FUNCTION_BLOCK FB_TXTDataExchanger IMPLEMENTS I_TXTDataExchanger
VAR CONSTANT
	iBUFFER_SIZE 						: UINT := 255;
END_VAR
VAR
	sName : STRING;
	
	(* First cycle bits used for selecting file logging mode *)
	bAddTimeStamp						: BOOL;
	bAddHeader							: BOOL;
	bCreateFileAtStart					: BOOL;    
                        		
	(* Internal status *)       		
	bActive 							: BOOL;										(*  *)
	bBusy								: BOOL;										(*  *)
	bError								: BOOL;										(*  *)
	iErrorID							: UDINT;									(*  *)
	                                                                            	
	eTXTDataExchangerState 				: E_TXTDataExchangerState;					(*  *)
	eTXTDataExchangerInitState 			: E_TXTDataExchangerInitState;				(*  *)
	eTXTDataExchangerAddLogsState		: E_TXTDataExchangerAddLogsState; 			(*  *)
	eTXTDataExchangerSetNewPathState 	: E_TXTDataExchangerSetNewPathState;
	eTXTDataExchangerSearchForFileState : E_TXTDataExchangerSearchForFileState;
	
	(* Internal parameters *)
	sFileName 							: STRING;									(*  *)
	sFileDir							: STRING;									(*  *)
	sFilePath							: STRING;									(*  *)
                   				      		
	hFile								: UINT;										(*  *)

	sAmsNetId							: T_AmsNetID;								(*  *)
	stTime								: TIMESTRUCT;								(*  *)
	sTime								: STRING;									(*  *)
	sFileDate							: STRING;									(*  *)

	sLogMessage							: STRING;									(*  *)

	sSearchFileName						: STRING; 
	bFileFound							: BOOL;                       		
	
	(* Buffer arrays *)         		
	iCurrentBufferLine					: UINT := 1;								(*  *)
	iCurrentBufferLineForFile			: UINT := 1;								(*  *)
	arrMessageBuffer 					: ARRAY [1..iBUFFER_SIZE] OF STRING(300);	(*  *)
	arrMessageBufferPresence			: ARRAY [1..iBUFFER_SIZE] OF BOOL(255);		(*  *)
	
	(* Function blocks - file handling *)
	fbFileOpen							: FB_FileOpen;								(*  *)
	fbFileClose							: FB_FileClose;								(*  *)
	fbCreateDir							: FB_CreateDir;								(*  *)
	fbFilePuts							: FB_FilePuts;								(*  *)
	fbEnumFindFileEntry					: FB_EnumFindFileEntry;
END_VAR

bActive := eTXTDataExchangerState >= TXT_DATA_EXCHANGER_READY;

IF fbMachineTime.bValid THEN
	stTime := fbMachineTime.systemTime;
	sTime := SYSTEMTIME_TO_STRING(stTime);
	
END_IF

StateMachine();

PROPERTY Active : REFERENCE TO BOOL
GET
Active REF= bActive;
END_GET
END_PROPERTY

PROPERTY AmsNetId : STRING
GET
AmsNetID := sAmsNetId;
END_GET
SET
sAmsNetId := AmsNetId;
END_SET
END_PROPERTY

PROPERTY Busy : REFERENCE TO BOOL
GET
Busy REF= bBusy;
END_GET
END_PROPERTY

PROPERTY Error : REFERENCE TO BOOL
GET
Error REF= bError;
END_GET
END_PROPERTY

PROPERTY ErrorID : REFERENCE TO UDINT
GET
ErrorID REF= iErrorID;
END_GET
END_PROPERTY

PROPERTY FileDir : STRING
GET
FileDir := sFileDir;
END_GET
SET
sFileDir := FileDir;
END_SET
END_PROPERTY

PROPERTY FileName : STRING
GET
FileName := sFileName;
END_GET
SET
sFileName := FileName;
END_SET
END_PROPERTY

METHOD M_ResetParameters : BOOL
VAR_INPUT
END_VAR
fbCreateDir( bExecute := FALSE);
fbFileOpen( bExecute := FALSE);
fbFilePuts( bExecute := FALSE);
fbFileClose( bExecute := FALSE);

FOR iCurrentBufferLine := 1 TO iBUFFER_SIZE BY 1 DO
	MEMSET(ADR(arrMessageBuffer[iCurrentBufferLine]),0,SIZEOF(arrMessageBuffer[iCurrentBufferLine]));
	arrMessageBufferPresence[iCurrentBufferLine] := FALSE;
END_FOR

iCurrentBufferLine := 1;
iCurrentBufferLineForFile := 1;

bError 		:= FALSE;
iErrorID 	:= 0;

MEMSET(ADR(sLogMessage),0,SIZEOF(sLogMessage));

eTXTDataExchangerInitState := 0;
eTXTDataExchangerAddLogsState := 0;
END_METHOD

METHOD M_SetNewPath : BOOL
VAR_INPUT
END_VAR
CASE eTXTDataExchangerSetNewPathState OF
	TXT_DATA_EXCHANGER_SET_NEW_PATH_CHANGE_PATH:
		M_SetNewPath := FALSE;
		sFilePath := FUN_MergeStrings3(sStr1 := sFileDir, sStr2 := sFileName, sStr3 :=  '.txt');
		eTXTDataExchangerSetNewPathState := TXT_DATA_EXCHANGER_SET_NEW_PATH_DONE;
	
	TXT_DATA_EXCHANGER_SET_NEW_PATH_DONE:
		M_SetNewPath := TRUE;
		eTXTDataExchangerSetNewPathState := TXT_DATA_EXCHANGER_SET_NEW_PATH_CHANGE_PATH;
			
END_CASE
END_METHOD

METHOD MR_Abort : BOOL
IF eTXTDataExchangerState >= TXT_DATA_EXCHANGER_READY THEN
	bBusy := TRUE;
	MR_Abort := FALSE;
	eTXTDataExchangerState := TXT_DATA_EXCHANGER_ABORTING;
	
ELSIF eTXTDataExchangerState = TXT_DATA_EXCHANGER_UNINITIALIZED THEN
	bBusy := FALSE;
	MR_Abort := TRUE;
	
END_IF
END_METHOD

METHOD MR_AddLogs : BOOL
VAR_INPUT
	sLogMessage 	: STRING;		
	
END_VAR
VAR
	sCurrentTime 	: STRING;
	sCurrentDate	: STRING;
	sLog			: STRING(300);
	
END_VAR
IF iCurrentBufferLine >= iBUFFER_SIZE THEN	
	iCurrentBufferLine := 1;
		
ELSE
	sCurrentDate := LEFT(sTime,10);
	sCurrentTime := RIGHT(sTime,12);
	MEMSET(ADR(sLog),0,SIZEOF(sLog));
	
	IF bAddTimeStamp THEN
		sLog := FUN_MergeStrings6(sCurrentDate,'$t',sCurrentTime,'$t',sLogMessage,'$n'); 
	ELSE
		sLog := CONCAT(sLogMessage,'$n'); 
	END_IF
	
	MEMSET(ADR(arrMessageBuffer[iCurrentBufferLine]),0,SIZEOF(arrMessageBuffer[iCurrentBufferLine]));
	arrMessageBuffer[iCurrentBufferLine] := sLog;
	iCurrentBufferLine := iCurrentBufferLine + 1;
	
	MR_AddLogs := TRUE;
	
END_IF
END_METHOD

METHOD MR_AddMESCommand : BOOL
VAR_INPUT
	sMachineID		: STRING;
	sOperatorID		: STRING;
	sPO				: STRING;
	sProductItem	: STRING;
	bLogOn			: BOOL;
END_VAR

VAR
	sLog			: STRING(300);
END_VAR
IF iCurrentBufferLine >= iBUFFER_SIZE THEN	
	iCurrentBufferLine := 1;
		
ELSE
	MEMSET(ADR(sLog),0,SIZEOF(sLog));

	IF bLogOn THEN
		sLog := FUN_MergeStrings10(sStr1 := 'DLG=A_P_AN|MNR=', 
									sStr2 := sMachineID,
									sStr3 := '|KNR=',
									sStr4 := sOperatorID,
									sStr5 := '|AUNR=',
									sStr6 := sPO,									
									sStr7 := '|ATK=',
									sStr8 := sProductItem,
									sStr9 := '|M_HS=1',
									sStr10 :='$n');  
									
	ELSE
		sLog := FUN_MergeStrings10(sStr1 := 'DLG=A_AB|MNR=', 
									sStr2 := sMachineID,
									sStr3 := '|KNR=',
									sStr4 := sOperatorID,
									sStr5 := '|AUNR=',
									sStr6 := sPO,									
									sStr7 := '|ATK=',
									sStr8 := sProductItem,
									sStr9 := '|M_HS=2',
									sStr10 :='$n');  
									
	END_IF
	
	MEMSET(ADR(arrMessageBuffer[iCurrentBufferLine]),0,SIZEOF(arrMessageBuffer[iCurrentBufferLine]));
	arrMessageBuffer[iCurrentBufferLine] := sLog;
	iCurrentBufferLine := iCurrentBufferLine + 1;
	
	MR_AddMESCommand := TRUE;
	
END_IF
END_METHOD

METHOD MR_FirstCycle : BOOL
VAR_INPUT
	sName 					: STRING;
	sFileDir				: STRING(255);
	sFileName				: STRING(255);
	sAmsNetId				: T_AmsNetID;		
	bAddTimeStamp			: BOOL;				(* If true the time stamp will be added to each log *)
	bAddHeader				: BOOL;				(* If true the header will be added to the file at the start-up *)
	bCreateFileAtStart		: BOOL;				(* If true the file will be created at the start-up *)
END_VAR
THIS^.sName := sName;
THIS^.sFileDir := sFileDir;
THIS^.sFileName := sFileName;
THIS^.sAmsNetId := sAmsNetId;
THIS^.bAddTimeStamp := bAddTimeStamp;
THIS^.bAddHeader := bAddHeader;
THIS^.bCreateFileAtStart := bCreateFileAtStart;

M_SetNewPath();
END_METHOD

METHOD MR_Init : BOOL
VAR_INPUT
END_VAR
IF eTXTDataExchangerState = TXT_DATA_EXCHANGER_UNINITIALIZED THEN
	bBusy := TRUE;
	MR_Init := FALSE;
	eTXTDataExchangerState := TXT_DATA_EXCHANGER_INITIALIZING;
	
ELSIF eTXTDataExchangerState >= TXT_DATA_EXCHANGER_READY THEN
	bBusy := FALSE;
	MR_Init := TRUE;
	
END_IF
END_METHOD

METHOD MR_Reset : BOOL
IF eTXTDataExchangerState >= TXT_DATA_EXCHANGER_IDLE AND eTXTDataExchangerState <> TXT_DATA_EXCHANGER_METHOD_DONE THEN
	bBusy := TRUE;
	MR_Reset := FALSE;
	eTXTDataExchangerState := TXT_DATA_EXCHANGER_RESET;	

ELSIF eTXTDataExchangerState = TXT_DATA_EXCHANGER_METHOD_DONE THEN
	bBusy := FALSE;
	MR_Reset := TRUE;

END_IF
END_METHOD

METHOD MR_SearchForFile : BOOL
VAR_INPUT
	sSearchFileName		: STRING;			(* Whole name of the search file (e.g.: "DemoFile.txt" *)
END_VAR

VAR_OUTPUT
	bFileFound	: BOOL;
END_VAR
IF eTXTDataExchangerState = TXT_DATA_EXCHANGER_IDLE THEN
	THIS^.sSearchFileName := sSearchFileName;
	bFileFound	:= FALSE;
	bBusy := TRUE;
	MR_SearchForFile := FALSE;
	eTXTDataExchangerState := TXT_DATA_EXCHANGER_SEARCH_FOR_FILE;
	
ELSIF eTXTDataExchangerState = TXT_DATA_EXCHANGER_METHOD_DONE THEN
	bFileFound := THIS^.bFileFound;
	bBusy := FALSE;
	MR_SearchForFile := TRUE;
	
END_IF
END_METHOD

METHOD MR_SelectPath : BOOL
VAR_INPUT
	sFileDir								: STRING; 			(* CSV source file directory name *)
	sFileName 								: STRING; 			(* CSV source file name *)
END_VAR
IF eTXTDataExchangerState = TXT_DATA_EXCHANGER_IDLE THEN
	THIS^.sFileDir := sFileDir;	
	THIS^.sFileName := sFileName;	
	bBusy := TRUE;
	MR_SelectPath := FALSE;
	eTXTDataExchangerState := TXT_DATA_EXCHANGER_SELECT_PATH;
	
ELSIF eTXTDataExchangerState = TXT_DATA_EXCHANGER_METHOD_DONE THEN
	bBusy := FALSE;
	MR_SelectPath := TRUE;
	
END_IF
END_METHOD

METHOD PROTECTED MS_Aborting
fbCreateDir( bExecute := FALSE);
fbFileOpen( bExecute := FALSE);
fbFilePuts( bExecute := FALSE);
fbFileClose( bExecute := FALSE);

FOR iCurrentBufferLine := 1 TO iBUFFER_SIZE BY 1 DO
	MEMSET(ADR(arrMessageBuffer[iCurrentBufferLine]),0,SIZEOF(arrMessageBuffer[iCurrentBufferLine]));
	arrMessageBufferPresence[iCurrentBufferLine] := FALSE;
	
END_FOR

iCurrentBufferLine := 1;
iCurrentBufferLineForFile := 1;

MEMSET(ADR(sTime),0,SIZEOF(sTime));
MEMSET(ADR(sFileDate),0,SIZEOF(sFileDate));
MEMSET(ADR(sLogMessage),0,SIZEOF(sLogMessage));

stTime.wDay 			:= 0;
stTime.wDayOfWeek 		:= 0;
stTime.wHour 			:= 0;
stTime.wMilliseconds 	:= 0;
stTime.wMinute 			:= 0;
stTime.wMonth 			:= 0;
stTime.wSecond 			:= 0;
stTime.wYear 			:= 0;

bActive		:= FALSE;
bBusy 		:= FALSE;
bError 		:= FALSE;
iErrorID 	:= 0;

eTXTDataExchangerInitState := TXT_DATA_EXCHANGER_INIT_GET_TIME;
eTXTDataExchangerAddLogsState := TXT_DATA_EXCHANGER_ADD_LOGS_OPEN;
eTXTDataExchangerState := TXT_DATA_EXCHANGER_UNINITIALIZED;
END_METHOD

METHOD PROTECTED MS_AddLogs
CASE eTXTDataExchangerAddLogsState OF
	TXT_DATA_EXCHANGER_ADD_LOGS_OPEN:
		IF NOT fbFileOpen.bError THEN
			fbFileOpen( sNetId 		:= sAmsNetId,
						sPathName 	:= sFilePath,
						bExecute 	:= TRUE,
						tTimeout	:= DEFAULT_ADS_TIMEOUT,
						nMode		:= FOPEN_MODEAPPEND OR FOPEN_MODEPLUS);
							
			IF NOT fbFileOpen.bBusy THEN
				fbFileOpen(bExecute := FALSE);				
				hFile := fbFileOpen.hFile;;
				eTXTDataExchangerAddLogsState := TXT_DATA_EXCHANGER_ADD_LOGS_WRITE;
			
			END_IF
		ELSE
			fbFileOpen( bExecute := FALSE);
			bError := fbFileOpen.bError;
			iErrorID := fbFileOpen.nErrId;

		END_IF
	

	TXT_DATA_EXCHANGER_ADD_LOGS_WRITE:
		IF NOT fbFilePuts.bError THEN
			fbFilePuts( sNetId		:= sAmsNetId,
						hFile 		:= hFile,
						sLine 		:= arrMessageBuffer[iCurrentBufferLineForFile],
						bExecute 	:= TRUE,
						tTimeout 	:= DEFAULT_ADS_TIMEOUT);	
					
			IF NOT fbFilePuts.bBusy THEN				
				eTXTDataExchangerAddLogsState := TXT_DATA_EXCHANGER_ADD_LOGS_WRITE_DONE;
				
			END_IF
			
		ELSE
			fbFilePuts( bExecute := FALSE);
			bError := fbFilePuts.bError;
			iErrorID := fbFilePuts.nErrId;
			
		END_IF	

		
	TXT_DATA_EXCHANGER_ADD_LOGS_WRITE_DONE:
		fbFilePuts( bExecute := FALSE);	
		iCurrentBufferLineForFile := iCurrentBufferLineForFile + 1;	
		
		IF iCurrentBufferLineForFile >= iBUFFER_SIZE THEN
			iCurrentBufferLineForFile := 1;
			
		ELSIF iCurrentBufferLineForFile < iCurrentBufferLine THEN
			eTXTDataExchangerAddLogsState := TXT_DATA_EXCHANGER_ADD_LOGS_WRITE;			
	
		ELSIF iCurrentBufferLineForFile >= iCurrentBufferLine THEN
			eTXTDataExchangerAddLogsState := TXT_DATA_EXCHANGER_ADD_LOGS_CLOSE;
			
		END_IF;

	
	TXT_DATA_EXCHANGER_ADD_LOGS_CLOSE:
		IF NOT fbFileClose.bError THEN
			fbFileClose(	sNetId := sAmsNetId,
							hFile := hFile,
							bExecute := TRUE,
							tTimeout := DEFAULT_ADS_TIMEOUT);
							
			IF NOT fbFileClose.bBusy THEN
				fbFileClose(bExecute := FALSE);
				eTXTDataExchangerAddLogsState := TXT_DATA_EXCHANGER_ADD_LOGS_OPEN;
				eTXTDataExchangerState := TXT_DATA_EXCHANGER_IDLE;

			END_IF
		ELSE
			bError := fbFileClose.bError;
			iErrorID := fbFileClose.nErrId;
			fbFileClose( bExecute := FALSE);
			
		END_IF
		
END_CASE
END_METHOD

METHOD PROTECTED MS_Idle
VAR_INPUT
END_VAR
IF iCurrentBufferLineForFile < iCurrentBufferLine THEN
	eTXTDataExchangerState := TXT_DATA_EXCHANGER_ADD_LOGS;

END_IF
END_METHOD

METHOD PROTECTED MS_Initializing //C:\TwinCAT\log\filelog.txt
CASE eTXTDataExchangerInitState OF
	TXT_DATA_EXCHANGER_INIT_CREATE_DIR:
		IF bCreateFileAtStart THEN
			fbCreateDir(sNetId 		:= sAmsNetId,
						sPathName 	:= sFileDir,
						bExecute 	:= TRUE,
						tTimeout 	:= DEFAULT_ADS_TIMEOUT);
						
			IF NOT fbCreateDir.bBusy THEN
				eTXTDataExchangerInitState := TXT_DATA_EXCHANGER_INIT_GET_TIME;
				fbCreateDir( bExecute := FALSE);
				
			END_IF
		ELSE
			eTXTDataExchangerInitState := TXT_DATA_EXCHANGER_INIT_DONE;
			
		END_IF
		
	TXT_DATA_EXCHANGER_INIT_GET_TIME:
		IF fbMachineTime.bValid THEN
			stTime := fbMachineTime.systemTime;
			sTime := SYSTEMTIME_TO_STRING(stTime);
			sFileDate := LEFT(sTime,10);
			eTXTDataExchangerInitState := TXT_DATA_EXCHANGER_INIT_CREATE_FILE;
			
		END_IF
		
	TXT_DATA_EXCHANGER_INIT_CREATE_FILE:
		IF NOT fbFileOpen.bError THEN
			fbFileOpen( sNetId 		:= sAmsNetId,
						sPathName 	:= sFilePath,
						bExecute 	:= TRUE,
						tTimeout	:= DEFAULT_ADS_TIMEOUT,
						nMode		:= FOPEN_MODEAPPEND OR FOPEN_MODEPLUS);
							
			IF NOT fbFileOpen.bBusy THEN
				hFile := fbFileOpen.hFile;
				fbFileOpen(bExecute := FALSE);		
				
				IF bAddHeader THEN 
					eTXTDataExchangerInitState := TXT_DATA_EXCHANGER_INIT_ADD_HEADER;
					
				ELSE
					eTXTDataExchangerInitState := TXT_DATA_EXCHANGER_INIT_CLOSE_FILE;
					
				END_IF							
			END_IF
		ELSE
			bError := fbFileOpen.bError;
			iErrorID := fbFileOpen.nErrId;
			fbFileOpen( bExecute := FALSE);
			
		END_IF
		
	TXT_DATA_EXCHANGER_INIT_ADD_HEADER:
		IF NOT fbFilePuts.bError THEN
			fbFilePuts(	sNetId := sAmsNetId,
						hFile := hFile,
						sLine := CONCAT('----- Logger file initialized at ',CONCAT(LEFT(sTime,23),' ----- $n')),
						bExecute := TRUE,
						tTimeout := DEFAULT_ADS_TIMEOUT);

			IF NOT fbFilePuts.bBusy THEN
				eTXTDataExchangerInitState := TXT_DATA_EXCHANGER_INIT_CLOSE_FILE;
				fbFilePuts( bExecute := FALSE);
				
			END_IF	
		ELSE
			bError := fbFilePuts.bError;
			iErrorID := fbFilePuts.nErrId;
			fbFilePuts( bExecute := FALSE);
			
		END_IF
	
	TXT_DATA_EXCHANGER_INIT_CLOSE_FILE:
		IF NOT fbFileClose.bError THEN
			fbFileClose( sNetId 		:= sAmsNetId,
							hFile 		:= hFile,
							bExecute 	:= TRUE,
							tTimeout 	:= DEFAULT_ADS_TIMEOUT);
							
			IF NOT fbFileClose.bBusy THEN
				eTXTDataExchangerInitState := TXT_DATA_EXCHANGER_INIT_DONE;
				fbFileClose( bExecute := FALSE);
				
			END_IF
		ELSE
			bError := fbFileClose.bError;
			iErrorID := fbFileClose.nErrId;
			fbFileClose( bExecute := FALSE);
			
		END_IF
	
	TXT_DATA_EXCHANGER_INIT_DONE:
		eTXTDataExchangerInitState := TXT_DATA_EXCHANGER_INIT_CREATE_DIR;
		eTXTDataExchangerState := TXT_DATA_EXCHANGER_IDLE;
		
END_CASE
END_METHOD

METHOD PROTECTED MS_MethodDone
VAR_INPUT
END_VAR
IF NOT bBusy THEN
	eTXTDataExchangerState := TXT_DATA_EXCHANGER_IDLE;

END_IF
END_METHOD

METHOD PROTECTED MS_Ready
VAR_INPUT
END_VAR
eTXTDataExchangerState := TXT_DATA_EXCHANGER_IDLE;
END_METHOD

METHOD PROTECTED MS_Reset
VAR_INPUT
END_VAR
IF M_ResetParameters() THEN
	eTXTDataExchangerState := TXT_DATA_EXCHANGER_METHOD_DONE;
	
END_IF
END_METHOD

METHOD MS_SearchForFile : BOOL
VAR_INPUT
END_VAR
CASE eTXTDataExchangerSearchForFileState OF
    TXT_DATA_EXCHANGER_SEARCH_FOR_FILE_ENUM_FIRST_ENTRY:
		bFileFound := FALSE;
		fbEnumFindFileEntry (sNetID := sAmsNetId, 
							 tTimeout := T#5S, 
							 sPathName := CONCAT(STR1 := sFileDir, STR2 := '*.*'));
		
		fbEnumFindFileEntry.eCmd := eEnumCmd_First;    (* enum first entry *)
		
		eTXTDataExchangerSearchForFileState := TXT_DATA_EXCHANGER_SEARCH_FOR_FILE_ENUM_NEXT_ENTRY;

    TXT_DATA_EXCHANGER_SEARCH_FOR_FILE_ENUM_NEXT_ENTRY:    (* enum one entry *)
        fbEnumFindFileEntry( bExecute := FALSE );
        fbEnumFindFileEntry( bExecute := TRUE );
		
        eTXTDataExchangerSearchForFileState := TXT_DATA_EXCHANGER_SEARCH_FOR_FILE_WAIT_FOR_READING;

    TXT_DATA_EXCHANGER_SEARCH_FOR_FILE_WAIT_FOR_READING:    (* wait until function block not busy *)
        fbEnumFindFileEntry( bExecute := FALSE );
		
        IF NOT fbEnumFindFileEntry.bBusy THEN
            IF NOT fbEnumFindFileEntry.bError THEN
                IF NOT fbEnumFindFileEntry.bEOE THEN
                   	IF sSearchFileName = fbEnumFindFileEntry.stFindFile.sFileName THEN
						bFileFound := TRUE;
						eTXTDataExchangerSearchForFileState := TXT_DATA_EXCHANGER_SEARCH_FOR_FILE_DONE;
						
					END_IF
                    fbEnumFindFileEntry.eCmd := eEnumCmd_Next; (* enum next entry *)
					
                    eTXTDataExchangerSearchForFileState := TXT_DATA_EXCHANGER_SEARCH_FOR_FILE_ENUM_NEXT_ENTRY;
					
                ELSE (* no more entries *)
                    eTXTDataExchangerSearchForFileState := TXT_DATA_EXCHANGER_SEARCH_FOR_FILE_DONE;
					
                END_IF
            ELSE (* log error *)       
				bError := fbEnumFindFileEntry.bError;
				iErrorID := fbEnumFindFileEntry.nErrID;
				eTXTDataExchangerSearchForFileState := TXT_DATA_EXCHANGER_SEARCH_FOR_FILE_DONE;
				
            END_IF
        END_IF
		
	TXT_DATA_EXCHANGER_SEARCH_FOR_FILE_DONE:
			eTXTDataExchangerSearchForFileState := TXT_DATA_EXCHANGER_SEARCH_FOR_FILE_ENUM_FIRST_ENTRY;
			eTXTDataExchangerState := TXT_DATA_EXCHANGER_METHOD_DONE;
		
END_CASE
END_METHOD

METHOD MS_SelectPath : BOOL
VAR_INPUT
END_VAR
IF M_SetNewPath() THEN
	eTXTDataExchangerState := TXT_DATA_EXCHANGER_METHOD_DONE;
	
END_IF
END_METHOD

METHOD PROTECTED MS_Uninitialized
;
END_METHOD

PROPERTY Name : STRING
GET
Name := sName;
END_GET
SET
sName := Name;
END_SET
END_PROPERTY

METHOD PROTECTED StateMachine
CASE eTXTDataExchangerState OF
	TXT_DATA_EXCHANGER_UNINITIALIZED:
		MS_Uninitialized();
		
	TXT_DATA_EXCHANGER_INITIALIZING:
		MS_Initializing();
		
	TXT_DATA_EXCHANGER_IDLE:
		MS_Idle();
		
	TXT_DATA_EXCHANGER_ADD_LOGS:
		MS_AddLogs();	
		
	TXT_DATA_EXCHANGER_SELECT_PATH:
		MS_SelectPath();			
		
	TXT_DATA_EXCHANGER_SEARCH_FOR_FILE:
		MS_SearchForFile();			
	
	TXT_DATA_EXCHANGER_RESET:
		MS_Reset();
		
	TXT_DATA_EXCHANGER_METHOD_DONE:
		MS_MethodDone();
	
	TXT_DATA_EXCHANGER_ABORTING:
		MS_Aborting();
	
END_CASE
END_METHOD

END_FUNCTION_BLOCK

(* stored: Version 1.1.0.1, ProductVersion 3.1.4024.9
   POU FB_TXTDataExchanger: Id {1a3ada84-04d4-4555-a76e-ba1e0f62a9de}, SpecialFunc None
   Folder FirstCycle: Id {1dd2ade0-cafa-4fdb-9516-ce06347d9323}
   Folder Internal: Id {237f2c8d-39bd-45e4-a467-94f9beb94055}
   Folder Properties: Id {ed94c300-77dd-4d6e-9b79-3098ed6f9fa7}
   Folder Parameters: Id {319916c7-d9d7-427f-86a9-2501160b1f87}
   Folder Status: Id {3771faaf-8ca4-46c1-bcbe-a06d00726d64}
   Folder Requests: Id {f24ad5f0-c66b-430d-b202-4b76428b888e}
   Folder StateMachine: Id {bd87b044-912f-4b85-bbb6-0052c7a5810c}
   Property Active: Id {ef71fc8b-26e1-4460-bfce-65a2005cc7b4}
   Get Get: Id {e3284859-0a8f-426b-8554-303b97e2fdd0}
   Property AmsNetId: Id {a57c9008-8f6d-46d6-ac3c-ad2896ec069e}
   Get Get: Id {64eb65ab-8e69-47d6-97bd-8b335cad7e18}
   Set Set: Id {de30aa7e-b6a2-4c61-964d-84d42d66dece}
   Property Busy: Id {5ad0da15-2b97-4188-9197-21f425c1fb39}
   Get Get: Id {611b1048-0a45-48b8-a8b6-e40ae9a9cfa1}
   Property Error: Id {30b73de8-fc64-426a-900d-fbb02d12cd7d}
   Get Get: Id {7fe8308d-4e5a-459e-bead-68837762acc8}
   Property ErrorID: Id {cf2a4bce-7e99-4df2-bdbf-2194c7985e51}
   Get Get: Id {cac29d90-5369-4273-8fed-b7dc894e32de}
   Property FileDir: Id {dbd902e6-860e-4d53-b0d0-72b8a054924f}
   Get Get: Id {fd60c011-e53f-434c-9294-c72e9ae3ad69}
   Set Set: Id {ca9c95c6-5a97-4c4c-ade2-35c2d24b0f9a}
   Property FileName: Id {bc042983-795c-4cb4-a333-d6444566baf9}
   Get Get: Id {1e668bcb-9986-4909-b994-9c42fcb71f6c}
   Set Set: Id {2d4d74d7-a6e5-49b2-ac33-54f00db52866}
   Method M_ResetParameters: Id {9a370994-42c4-4f1c-b077-4efbcd9f2e53}
   Method M_SetNewPath: Id {92d1eb7b-cedc-423b-9025-3187ac31c19c}
   Method MR_Abort: Id {631c74f0-7146-4340-b4a4-6b79b406d46e}
   Method MR_AddLogs: Id {6fd86b1b-ab07-4f96-9b44-cf3b33aea90a}
   Method MR_AddMESCommand: Id {dd4df726-842d-4d70-a31b-5fbeeb375aeb}
   Method MR_FirstCycle: Id {b89de474-da9f-443e-b1b1-a5c45d17d08e}
   Method MR_Init: Id {18370ca5-11a1-4371-b8fa-f305110c19d0}
   Method MR_Reset: Id {d565da08-4dc2-45d6-a9f1-7094c275eea6}
   Method MR_SearchForFile: Id {e98733aa-949c-4b7e-b0c5-39542333ad93}
   Method MR_SelectPath: Id {35634623-aa82-428f-8665-abd18b4cf7af}
   Method MS_Aborting: Id {6abc35c7-e046-42b2-a411-30f9fb36de79}
   Method MS_AddLogs: Id {a77aba60-7e24-4b64-bbdf-2d910dd5d63c}
   Method MS_Idle: Id {db1bc726-252f-4c03-aa4d-9e25c54fc7e2}
   Method MS_Initializing: Id {14e1fde6-1d3a-4806-8cd1-6eab3ea9b532}
   Method MS_MethodDone: Id {2f3fd77c-c6ee-4a6e-8cfb-79b7ecd1c52b}
   Method MS_Ready: Id {e18836d8-72f2-47a8-97b3-1fe6b1c659db}
   Method MS_Reset: Id {fb5d8fc6-5068-4e3e-94b6-f28af10d6aac}
   Method MS_SearchForFile: Id {d5869d26-d7d9-4d2f-9cb7-73b2d86f9cb7}
   Method MS_SelectPath: Id {4fb457ee-747b-41e1-a5f7-8fbe8f662bae}
   Method MS_Uninitialized: Id {a2dbf8a9-4867-41f8-b176-07f2375a7b52}
   Property Name: Id {37d6402b-4711-420d-8da0-ef91dc38d80d}
   Get Get: Id {d090d2fb-84ad-4b4b-a9cd-7c2b1e67d897}
   Set Set: Id {3eea3c8c-f2fa-4faa-bfae-67339695a1ff}
   Method StateMachine: Id {b3b23c31-97e9-4c87-8c8c-7c47bcaf2578} *)
